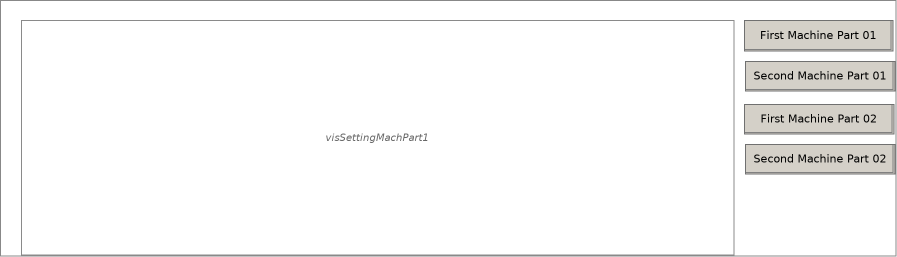
VISUALIZATION visMain  // 897x257
VAR_IN_OUT
	
END_VAR
VAR
	nSel : INT := 0;
END_VAR
    Frame (21,20 713x235)
        shows visSettingMachPart1(refSetting := MAIN.fbMach01_1.pSettings^)
        shows visSettingMachPart1(refSetting := MAIN.fbMach01_2.pSettings^)
        shows visSettingMachPart2(refSetting := MAIN.fbMach02_1.pSettings^)
        shows visSettingMachPart2(refSetting := MAIN.fbMach02_2.pSettings^)
    Button (744,20 149x31), "First Machine Part 01", colour toggle: nSel = 0
        OnMouseClick: FrameSelectionChange Selection=SelectedFrame=4000cae3-cddb-40df-befc-2ce2e2612873, GlobSel=AssignType=Directly, SelType=Locally
        OnMouseClick: execute { nSel := 0; }
    Button (745,61 150x30), "Second Machine Part 01", colour toggle: nSel = 1
        OnMouseClick: FrameSelectionChange Selection=SelectedFrame=4000cae3-cddb-40df-befc-2ce2e2612873, Selection=1, GlobSel=AssignType=Directly, SelType=Locally
        OnMouseClick: execute { nSel := 1; }
    Button (744,104 150x30), "First Machine Part 02", colour toggle: nSel = 2
        OnMouseClick: FrameSelectionChange Selection=SelectedFrame=4000cae3-cddb-40df-befc-2ce2e2612873, Selection=2, GlobSel=AssignType=Directly, SelType=Locally
        OnMouseClick: execute { nSel := 2; }
    Button (745,144 150x30), "Second Machine Part 02", colour toggle: nSel = 3
        OnMouseClick: FrameSelectionChange Selection=SelectedFrame=4000cae3-cddb-40df-befc-2ce2e2612873, Selection=3, GlobSel=AssignType=Directly, SelType=Locally
        OnMouseClick: execute { nSel := 3; }
END_VISUALIZATION

(* stored: Version 1.1.0.1, ProductVersion 3.1.4019.2
   Visu visMain: Id {7981d6cb-74da-404b-bace-db9241e6cb3e} *)
